// TwinCAT 3 PLC project VacuumPLC
// ProgramVersion: 3.1.4024.0
// libraries:
//   Tc2_Standard, * (Beckhoff Automation GmbH)
//   Tc2_System, * (Beckhoff Automation GmbH)
//   Tc3_Module, * (Beckhoff Automation GmbH)
// project tree:
//   DUTs/ Loader.TcDUT, Pump.TcDUT
//   GVLs/ GVL.TcGVL
//   / PlcTask.TcTTO
//   POUs/ Alarms.TcPOU, Common_Pulses.TcPOU, HMI.TcPOU, MAIN.TcPOU, Loaders.TcPOU, Pumps.TcPOU
//   POUs/Blocks and Functions/ BitCounter.TcPOU (not stored), FB_Loader.TcPOU
// real-time tasks:
//   TASK PlcTask: cycle T#10ms, priority 20, ADS port 350
// I/O:
//   DEVICE Device 2 (EtherCAT), AmsNetId 192.168.250.42.3.1
//     Term 5 (EK1200) [EK1200-5000 EtherCAT Power supply (2A E-Bus)]
//       Term 6 (EL3064) [EL3064 4Ch. Ana. Input 0-10V]
//       Term 7 (EL4002) [EL4002 2Ch. Ana. Output 0-10V, 12bit]
//       Term 8 (EL1889) [EL1889 16Ch. Dig. Input 24V, 3ms, negative]
//       Term 9 (EL2889) [EL2889 16Ch. Dig. Output 24V, 0.5A, negative]
//       Term 10 (EL6021) [EL6021 Interface (RS422/485)]
//       Term 11 (EK1122) [EK1122 2 port EtherCAT junction]
//       Term 12 (EL9011) [EL9011 End Terminal]
// variable links:
//   VacuumPLC/VacuumPLC Instance <-> Device 2 (EtherCAT)/Term 5 (EK1200)/Term 8 (EL1889)
//     PlcTask Inputs/Loaders.Loader_1.Flap_Reed <-> Channel 4/Input
//     PlcTask Inputs/Loaders.Loader_1.Level_Prox <-> Channel 3/Input
//     PlcTask Inputs/Loaders.Loader_1.Switch <-> Channel 5/Input
//     PlcTask Inputs/Pumps.Pump_1.Over_Load <-> Channel 2/Input
//     PlcTask Inputs/Pumps.Pump_1.Switch <-> Channel 1/Input
//   VacuumPLC/VacuumPLC Instance <-> Device 2 (EtherCAT)/Term 5 (EK1200)/Term 9 (EL2889)
//     PlcTask Outputs/Loaders.Loader_1.Valve <-> Channel 7/Output
//     PlcTask Outputs/Pumps.Pump_1.Join_Valve <-> Channel 6/Output
//     PlcTask Outputs/Pumps.Pump_1.Lamp <-> Channel 1/Output
//     PlcTask Outputs/Pumps.Pump_1.Line_Block <-> Channel 5/Output
//     PlcTask Outputs/Pumps.Pump_1.Motor <-> Channel 2/Output
//     PlcTask Outputs/Pumps.Pump_1.Pump_Block <-> Channel 3/Output
//     PlcTask Outputs/Pumps.Pump_1.Pump_Vent <-> Channel 4/Output

CONFIGURATION VacuumPLC
    RESOURCE PLC ON TwinCAT3
        TASK PlcTask(INTERVAL := T#10ms, PRIORITY := 20);
        PROGRAM MAIN WITH PlcTask : MAIN;
    END_RESOURCE
END_CONFIGURATION

// ---- DUTs/Loader.TcDUT
TYPE Loader :
STRUCT
	Level_Prox AT%I* : BOOL;
	Flap_Reed AT%I* : BOOL;
	Switch AT%I* : BOOL;
	PushButton AT%I* : BOOL;
	Valve AT%Q* : BOOL;
	Lamp AT%Q* : BOOL;
	Status_Word : WORD;
	HMI_Status_Word : WORD;
END_STRUCT
END_TYPE

// ---- DUTs/Pump.TcDUT
TYPE Pump :
STRUCT
	Switch AT%I* : BOOL;
	Over_Load AT%I* : BOOL;
	Lamp AT%Q* : BOOL;
	Motor AT%Q* : BOOL;
	Pump_Block AT%Q* : BOOL;
	Pump_Vent AT%Q* : BOOL;
	Line_Block AT%Q* : BOOL;
	Join_Valve AT%Q* : BOOL;
	{attribute 'OPC.UA.DA' := '1'}
	Status_Word : WORD;
	Rest_Time : CTU;
	Off_Delay : TON;
	Clean_On : CTU;
	Air_Delay : TON;
	Steady : TON;
	Conv_End : CTU;
	Max_Conv_Time : TON;
	Max_Conv_Time_ET : TIME;
	Min_Conv_Time : TON;
	Accumulated_Time : DINT;
	Efficency : INT;
	Temp_Accum_Time : INT;
	Locel_Request : BOOL;
	Global_Request : BOOL;
	Global_Grant : BOOL;
	Line_Live : BOOL;
	Locked_1 : BOOL;
	Locked_2 : BOOL;
	START_Conv : BOOL;
	LOCK_Start : BOOL;
	AUTO_Clean : BOOL;
	PumpOnDifu  : BOOL;
	Top_prox_OK : BOOL;
	Auto_Clean_Keep : SR;
	Pump_Block_Keep : SR;
	Locked_2_Keep : RS;
	Motor_Keep : RS;
	Scanner : INT;
	Pump_Requests : INT;
	Lock_Start_DIFU : R_TRIG;
	Conv_Start_DIFU : R_TRIG;
	Max_Conv_Time_PT : TIME; 
	Vac_Req_Sum : UINT;
	Vac_Req_Size : UINT := 32;
	Clean_Delay_PV : UINT := 300; //Use this VAR to be able to change when needs to initiate auto clean before shot down
	Clean_Delay_CV : INT := 300;
	Clean_Delay_Keep : SR;
	Clean_Delay_DIFU : R_TRIG;
END_STRUCT
END_TYPE

// ---- GVLs/GVL.TcGVL
//{attribute 'qualified_only'}
VAR_GLOBAL
	Always_ON : BOOL := 1;
	Vacuum_Grants : ARRAY [0..31] OF BOOL;
	Vacuum_Requests : ARRAY [0..31] OF BOOL;
	Conv_Max_Times : ARRAY [0..31] OF DWORD := [32(30000)];
	Conv_Last_Times : ARRAY [0..31] OF DWORD;
	testvar : WORD;
END_VAR

// ---- POUs/MAIN.TcPOU
PROGRAM MAIN
VAR
END_VAR

// To activate a section in the progem it has to be written in the MAIN (PRG). the sequence of the sections would determine what run first in the progrem.
Common_Pulses();
Pumps();
Loaders();
Alarms();
	GVL.testvar := Pumps.Pump_1.Status_Word;

END_PROGRAM

// ---- POUs/Common_Pulses.TcPOU
PROGRAM Common_Pulses
VAR
	Timer_0_1_s : TON;		// 0.1 seconds pulse
	Timer_1_0_s : TON;		// 1.0 seconds pulse
	Timer_1_0_m : TON;		// 1.0 minutes pulse
	Timer_10_0_m : TON;		// 10.0 minutes pulse
	Timer0_5_s_ON : TON;	// 0.5 second TON for 1 second blink like P_1_0 from CJ
	Timer0_5_s_OFF : TOF;	// 0.5 second TOF for 1 second blink like P_1_0 from CJ
	Timer_50_ms_ON : TON;	// 50 mili second TON for 0.1 second blink like P_0_1 from CJ
	Timer_50_ms_OFF : TOF;	// 50 mili second TOF for 0.1 second blink like P_0_1 from CJ
	Blink_1_s : BOOL;		// 1 second blink for lamp when ON
	Blink_0_1_s : BOOL;		// 0.1 second blink for lamp when alarm
END_VAR

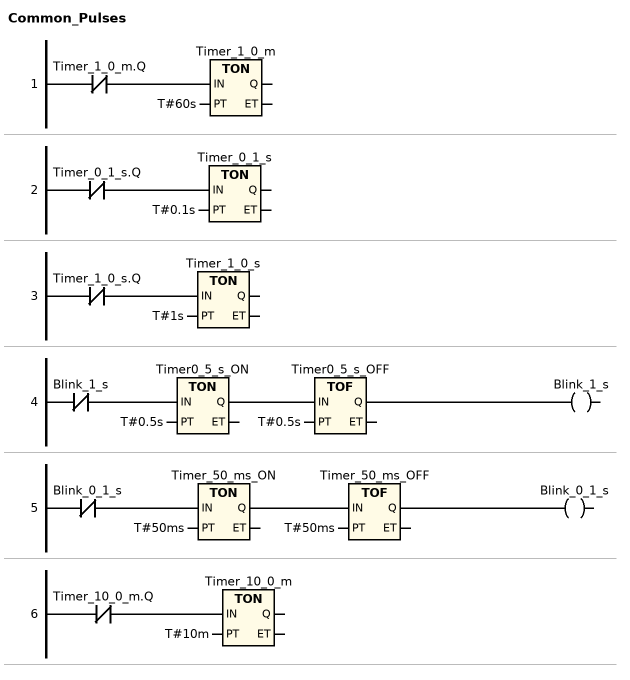
// NETWORK 1
Timer_1_0_m(IN := NOT Timer_1_0_m.Q, PT := T#60s); // TON

// NETWORK 2
Timer_0_1_s(IN := NOT Timer_0_1_s.Q, PT := T#0.1s); // TON

// NETWORK 3
Timer_1_0_s(IN := NOT Timer_1_0_s.Q, PT := T#1s); // TON

// NETWORK 4
Timer0_5_s_ON(IN := NOT Blink_1_s, PT := T#0.5s); // TON
Timer0_5_s_OFF(IN := Timer0_5_s_ON.Q, PT := T#0.5s); // TOF
Blink_1_s := Timer0_5_s_OFF.Q;

// NETWORK 5
Timer_50_ms_ON(IN := NOT Blink_0_1_s, PT := T#50ms); // TON
Timer_50_ms_OFF(IN := Timer_50_ms_ON.Q, PT := T#50ms); // TOF
Blink_0_1_s := Timer_50_ms_OFF.Q;

// NETWORK 6
Timer_10_0_m(IN := NOT Timer_10_0_m.Q, PT := T#10m); // TON

END_PROGRAM

// ---- POUs/Pumps.TcPOU
PROGRAM Pumps
VAR
	Pump_1 : Pump;
END_VAR
VAR // added by the converter: edge detectors and wires of the graphical bodies
    _w1, _w2, _w3, _w4, _w5, _w6, _w7, _w8, _w9 : BOOL;
END_VAR

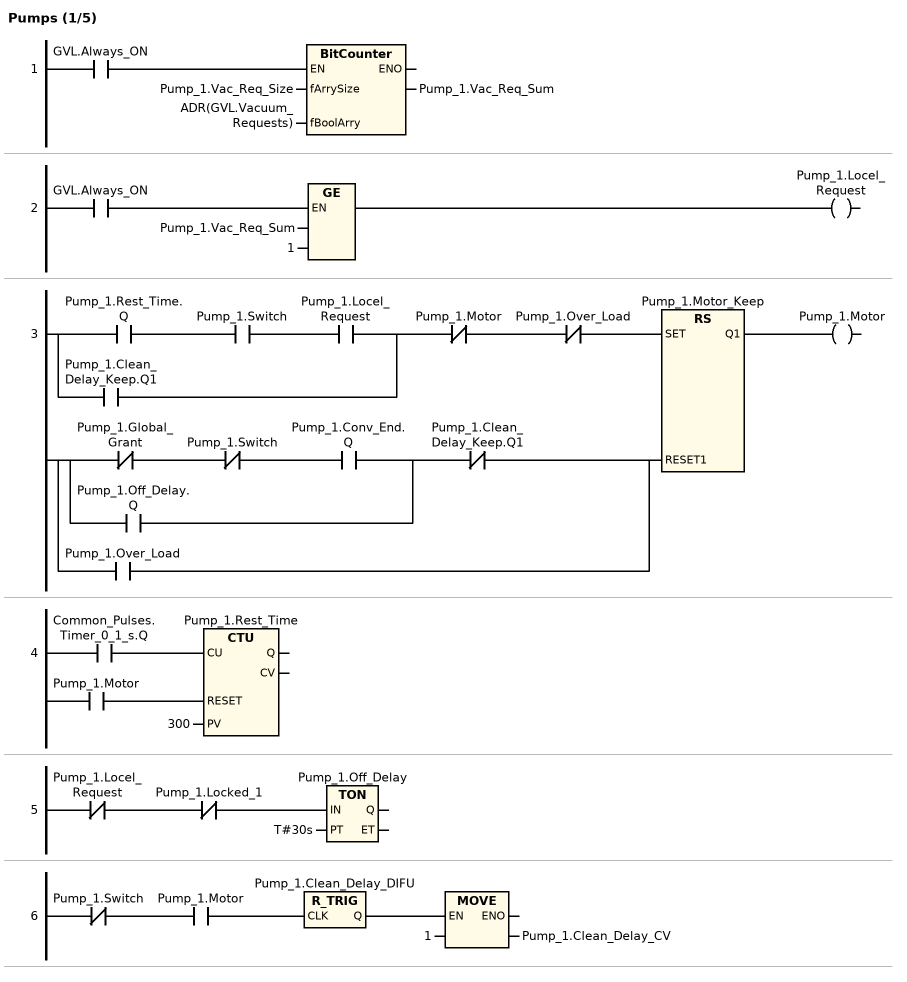
// NETWORK 1
IF GVL.Always_ON THEN
    Pump_1.Vac_Req_Sum := BitCounter(fArrySize := Pump_1.Vac_Req_Size, fBoolArry := ADR(GVL.Vacuum_Requests));
END_IF

// NETWORK 2
Pump_1.Locel_Request := GVL.Always_ON AND Pump_1.Vac_Req_Sum >= 1;

// NETWORK 3
Pump_1.Motor_Keep(SET := (Pump_1.Rest_Time.Q AND Pump_1.Switch AND Pump_1.Locel_Request OR Pump_1.Clean_Delay_Keep.Q1) AND NOT Pump_1.Motor AND NOT Pump_1.Over_Load, RESET1 := (NOT Pump_1.Global_Grant AND NOT Pump_1.Switch AND Pump_1.Conv_End.Q OR Pump_1.Off_Delay.Q) AND NOT Pump_1.Clean_Delay_Keep.Q1 OR Pump_1.Over_Load); // RS
Pump_1.Motor := Pump_1.Motor_Keep.Q1;

// NETWORK 4
Pump_1.Rest_Time(CU := Common_Pulses.Timer_0_1_s.Q, RESET := Pump_1.Motor, PV := 300); // CTU

// NETWORK 5
Pump_1.Off_Delay(IN := NOT Pump_1.Locel_Request AND NOT Pump_1.Locked_1, PT := T#30s); // TON

// NETWORK 6
Pump_1.Clean_Delay_DIFU(CLK := NOT Pump_1.Switch AND Pump_1.Motor); // R_TRIG
IF Pump_1.Clean_Delay_DIFU.Q THEN Pump_1.Clean_Delay_CV := 1; END_IF

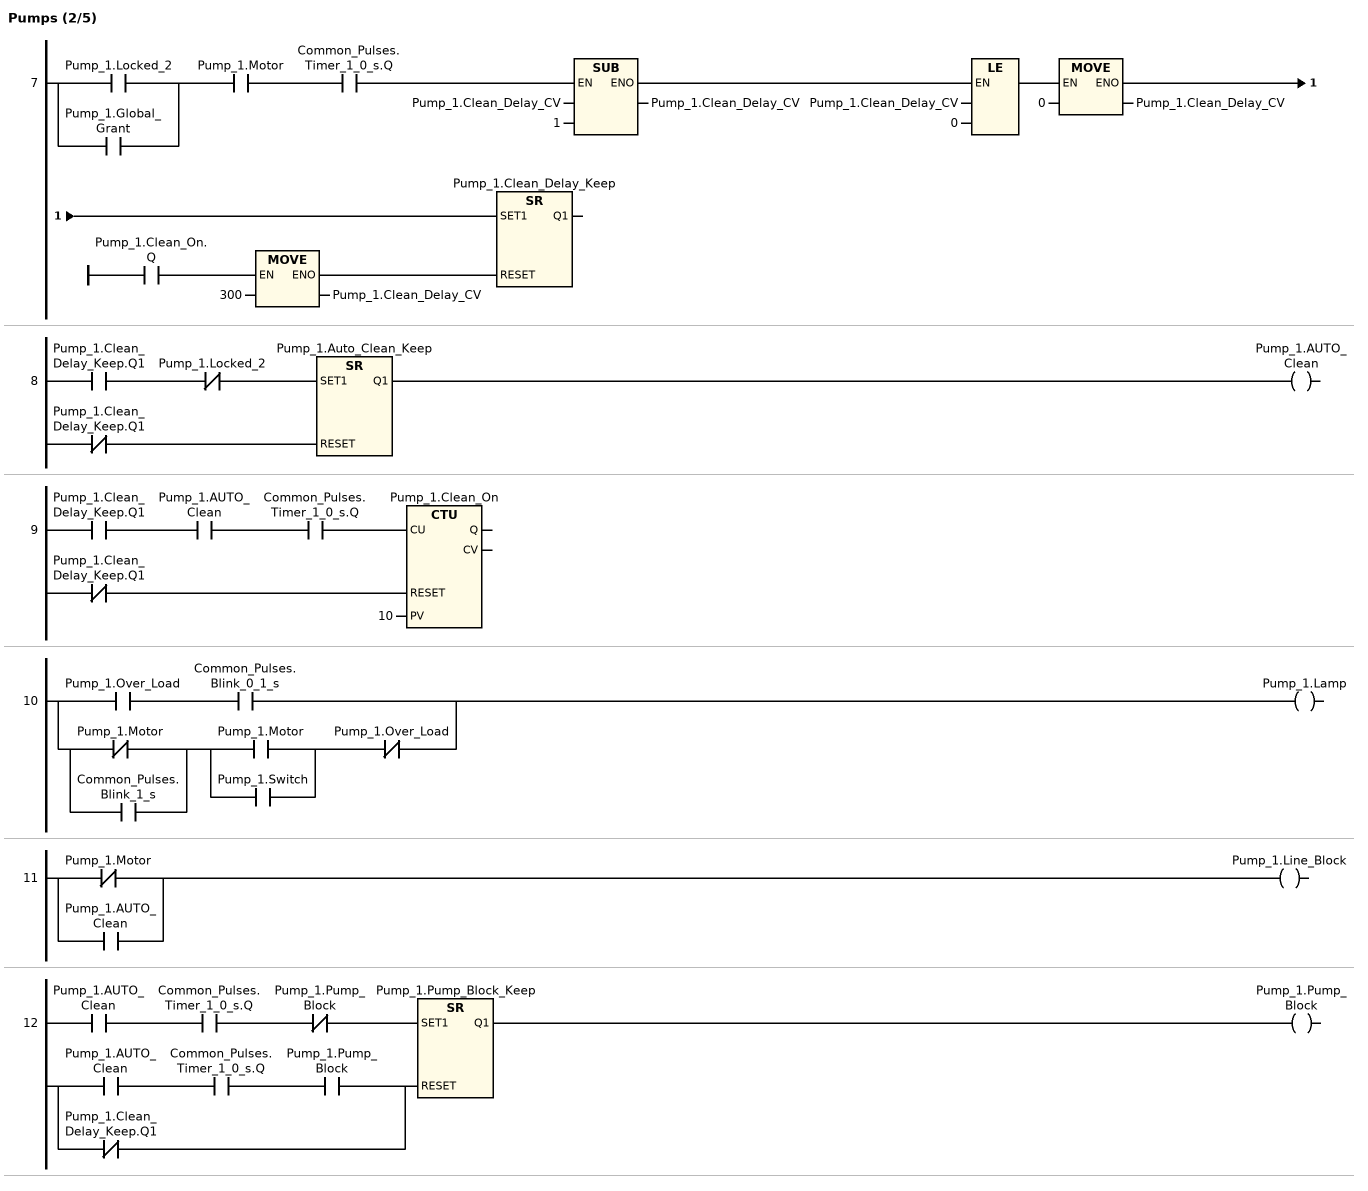
// NETWORK 7
_w1 := (Pump_1.Locked_2 OR Pump_1.Global_Grant) AND Pump_1.Motor AND Common_Pulses.Timer_1_0_s.Q;
IF _w1 THEN Pump_1.Clean_Delay_CV := Pump_1.Clean_Delay_CV - 1; END_IF
IF _w1 AND Pump_1.Clean_Delay_CV <= 0 THEN Pump_1.Clean_Delay_CV := 0; END_IF
_w3 := _w1 AND Pump_1.Clean_Delay_CV <= 0;
_w2 := Pump_1.Clean_On.Q;
IF _w2 THEN Pump_1.Clean_Delay_CV := 300; END_IF
Pump_1.Clean_Delay_Keep(SET1 := _w3, RESET := _w2); // SR

// NETWORK 8
Pump_1.Auto_Clean_Keep(SET1 := Pump_1.Clean_Delay_Keep.Q1 AND NOT Pump_1.Locked_2, RESET := NOT Pump_1.Clean_Delay_Keep.Q1); // SR
Pump_1.AUTO_Clean := Pump_1.Auto_Clean_Keep.Q1;

// NETWORK 9
Pump_1.Clean_On(
    CU := Pump_1.Clean_Delay_Keep.Q1 AND Pump_1.AUTO_Clean AND Common_Pulses.Timer_1_0_s.Q,
    RESET := NOT Pump_1.Clean_Delay_Keep.Q1,
    PV := 10); // CTU

// NETWORK 10
Pump_1.Lamp := Pump_1.Over_Load AND Common_Pulses.Blink_0_1_s OR (NOT Pump_1.Motor OR Common_Pulses.Blink_1_s) AND (Pump_1.Motor OR Pump_1.Switch) AND NOT Pump_1.Over_Load;

// NETWORK 11
Pump_1.Line_Block := NOT Pump_1.Motor OR Pump_1.AUTO_Clean;

// NETWORK 12
Pump_1.Pump_Block_Keep(SET1 := Pump_1.AUTO_Clean AND Common_Pulses.Timer_1_0_s.Q AND NOT Pump_1.Pump_Block, RESET := Pump_1.AUTO_Clean AND Common_Pulses.Timer_1_0_s.Q AND Pump_1.Pump_Block OR NOT Pump_1.Clean_Delay_Keep.Q1); // SR
Pump_1.Pump_Block := Pump_1.Pump_Block_Keep.Q1;

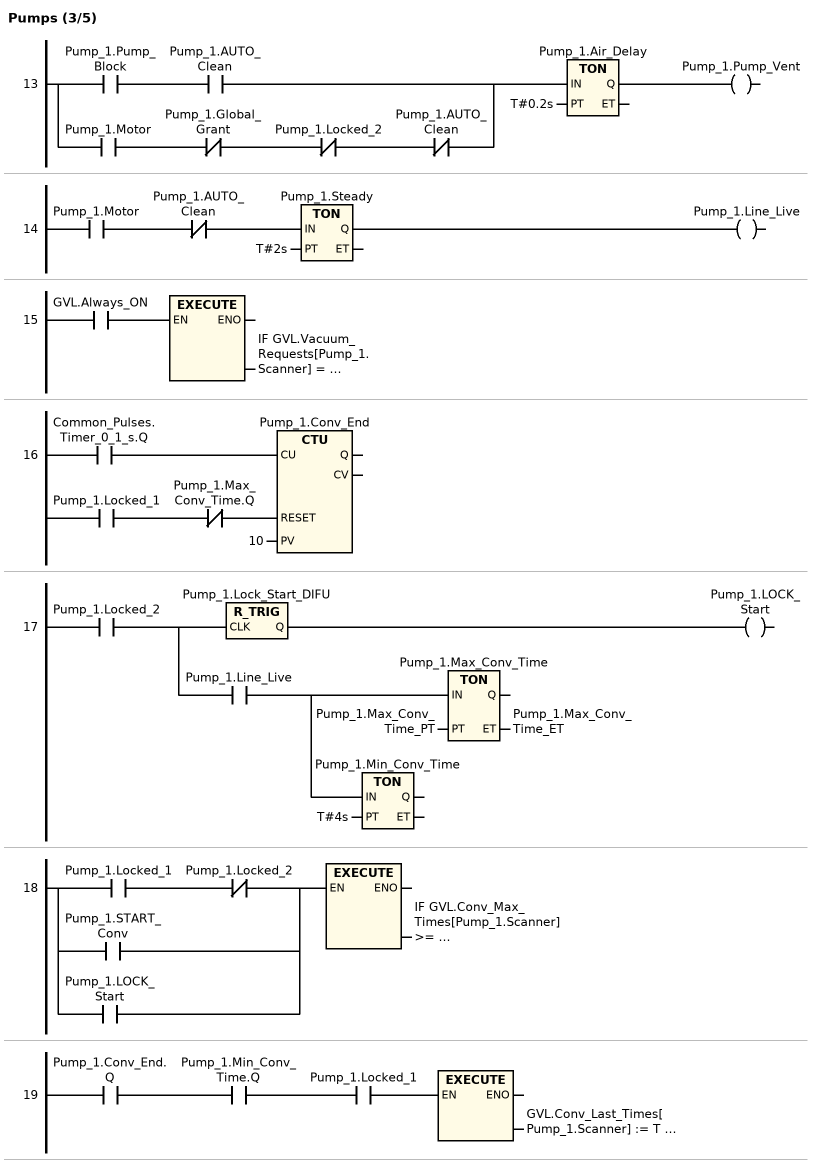
// NETWORK 13
Pump_1.Air_Delay(IN := Pump_1.Pump_Block AND Pump_1.AUTO_Clean OR Pump_1.Motor AND NOT Pump_1.Global_Grant AND NOT Pump_1.Locked_2 AND NOT Pump_1.AUTO_Clean, PT := T#0.2s); // TON
Pump_1.Pump_Vent := Pump_1.Air_Delay.Q;

// NETWORK 14
Pump_1.Steady(IN := Pump_1.Motor AND NOT Pump_1.AUTO_Clean, PT := T#2s); // TON
Pump_1.Line_Live := Pump_1.Steady.Q;

// NETWORK 15
IF GVL.Always_ON THEN
    IF GVL.Vacuum_Requests[Pump_1.Scanner] = 1 THEN 
    	Pump_1.Locked_1 := TRUE;
    	ELSE Pump_1.Locked_1 := FALSE;
    END_IF
END_IF

// NETWORK 16
Pump_1.Conv_End(
    CU := Common_Pulses.Timer_0_1_s.Q,
    RESET := Pump_1.Locked_1 AND NOT Pump_1.Max_Conv_Time.Q,
    PV := 10); // CTU

// NETWORK 17
Pump_1.Lock_Start_DIFU(CLK := Pump_1.Locked_2); // R_TRIG
Pump_1.LOCK_Start := Pump_1.Lock_Start_DIFU.Q;
_w4 := Pump_1.Locked_2 AND Pump_1.Line_Live;
Pump_1.Max_Conv_Time(IN := _w4, PT := Pump_1.Max_Conv_Time_PT, ET => Pump_1.Max_Conv_Time_ET); // TON
Pump_1.Min_Conv_Time(IN := _w4, PT := T#4s); // TON

// NETWORK 18
IF Pump_1.Locked_1 AND NOT Pump_1.Locked_2 OR Pump_1.START_Conv OR Pump_1.LOCK_Start THEN
    IF GVL.Conv_Max_Times[Pump_1.Scanner] >= 5000 THEN
    	Pump_1.Max_Conv_Time_PT := DWORD_TO_TIME(GVL.Conv_Max_Times[Pump_1.Scanner]);
    	ELSE Pump_1.Max_Conv_Time.PT := T#5S;
    END_IF
END_IF

// NETWORK 19
IF Pump_1.Conv_End.Q AND Pump_1.Min_Conv_Time.Q AND Pump_1.Locked_1 THEN
    GVL.Conv_Last_Times[Pump_1.Scanner] := TIME_TO_DWORD(Pump_1.Max_Conv_Time.ET);
    MEMSET (destAddr := ADR(GVL.Vacuum_Requests), fillByte := 0, n := SIZEOF(GVL.Vacuum_Requests));
END_IF

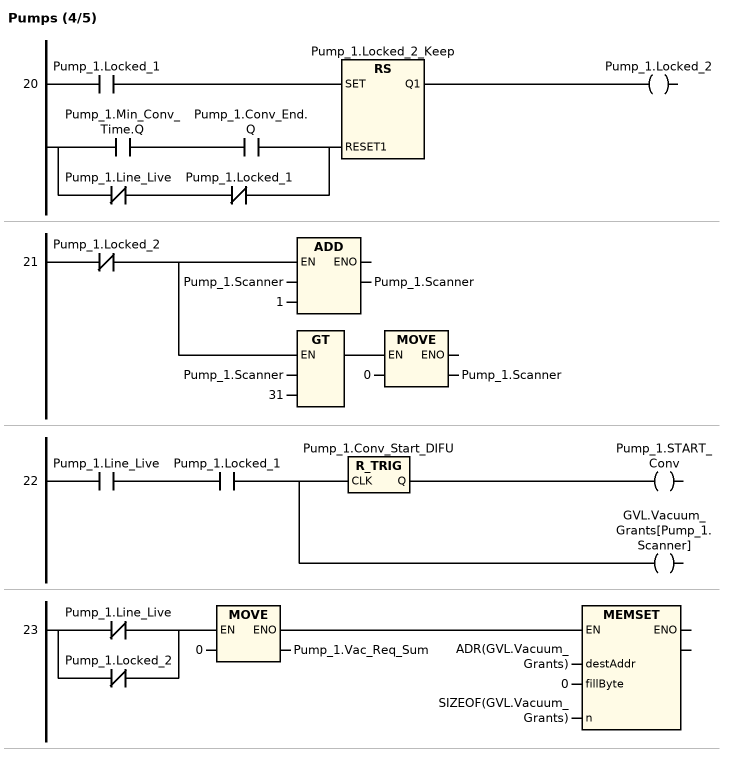
// NETWORK 20
Pump_1.Locked_2_Keep(SET := Pump_1.Locked_1, RESET1 := Pump_1.Min_Conv_Time.Q AND Pump_1.Conv_End.Q OR NOT Pump_1.Line_Live AND NOT Pump_1.Locked_1); // RS
Pump_1.Locked_2 := Pump_1.Locked_2_Keep.Q1;

// NETWORK 21
_w5 := NOT Pump_1.Locked_2;
IF _w5 THEN Pump_1.Scanner := Pump_1.Scanner + 1; END_IF
IF _w5 AND Pump_1.Scanner > 31 THEN Pump_1.Scanner := 0; END_IF

// NETWORK 22
_w6 := Pump_1.Line_Live AND Pump_1.Locked_1;
Pump_1.Conv_Start_DIFU(CLK := _w6); // R_TRIG
Pump_1.START_Conv := Pump_1.Conv_Start_DIFU.Q;
GVL.Vacuum_Grants[Pump_1.Scanner] := _w6;

// NETWORK 23
_w7 := NOT Pump_1.Line_Live OR NOT Pump_1.Locked_2;
IF _w7 THEN Pump_1.Vac_Req_Sum := 0; END_IF
IF _w7 THEN MEMSET(destAddr := ADR(GVL.Vacuum_Grants), fillByte := 0, n := SIZEOF(GVL.Vacuum_Grants)); END_IF

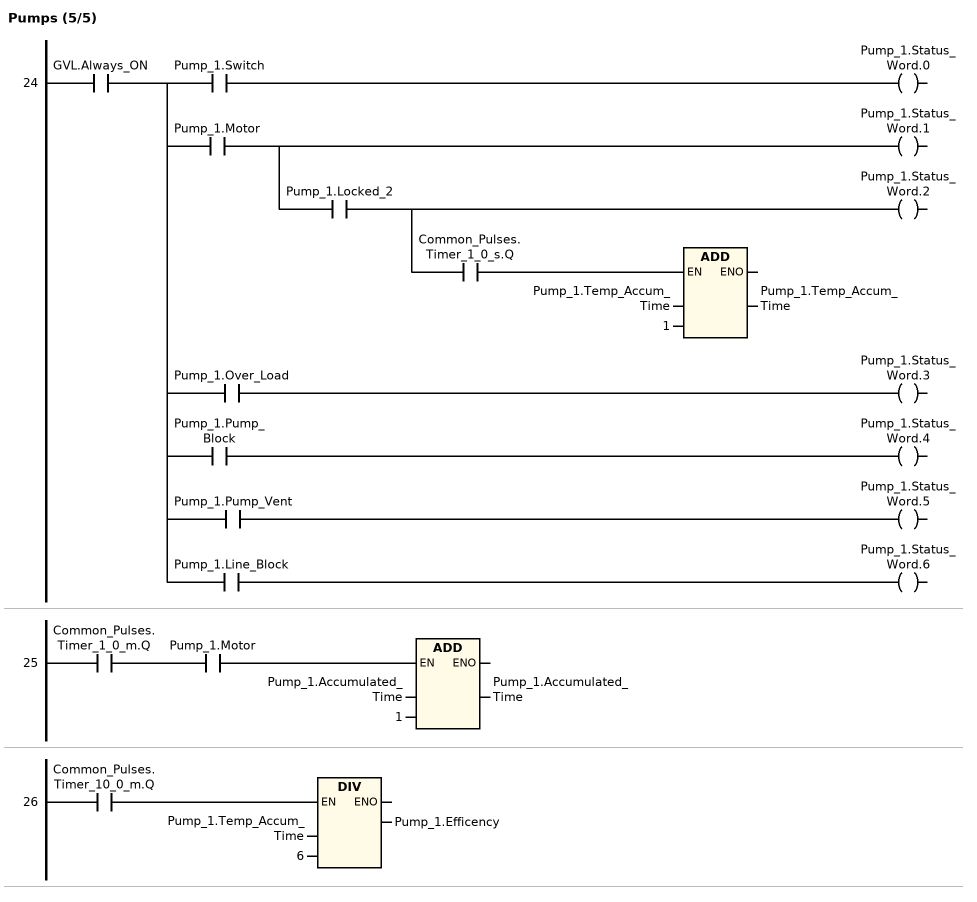
// NETWORK 24
Pump_1.Status_Word.0 := GVL.Always_ON AND Pump_1.Switch;
_w8 := GVL.Always_ON AND Pump_1.Motor;
Pump_1.Status_Word.1 := _w8;
_w9 := _w8 AND Pump_1.Locked_2;
Pump_1.Status_Word.2 := _w9;
IF _w9 AND Common_Pulses.Timer_1_0_s.Q THEN Pump_1.Temp_Accum_Time := Pump_1.Temp_Accum_Time + 1; END_IF
Pump_1.Status_Word.3 := GVL.Always_ON AND Pump_1.Over_Load;
Pump_1.Status_Word.4 := GVL.Always_ON AND Pump_1.Pump_Block;
Pump_1.Status_Word.5 := GVL.Always_ON AND Pump_1.Pump_Vent;
Pump_1.Status_Word.6 := GVL.Always_ON AND Pump_1.Line_Block;

// NETWORK 25
IF Common_Pulses.Timer_1_0_m.Q AND Pump_1.Motor THEN Pump_1.Accumulated_Time := Pump_1.Accumulated_Time + 1; END_IF

// NETWORK 26
IF Common_Pulses.Timer_10_0_m.Q THEN Pump_1.Efficency := Pump_1.Temp_Accum_Time / 6; END_IF

END_PROGRAM

// ---- POUs/Loaders.TcPOU
PROGRAM Loaders
VAR
	Loader_1: Loader;
	Loader_2: Loader;
	Loader_3: Loader;
	FB_Loader_1: FB_Loader;
	FB_Loader_2: FB_Loader;
	FB_Loader_3: FB_Loader;
END_VAR

// note: this text did not pass the execution check against the stored diagram
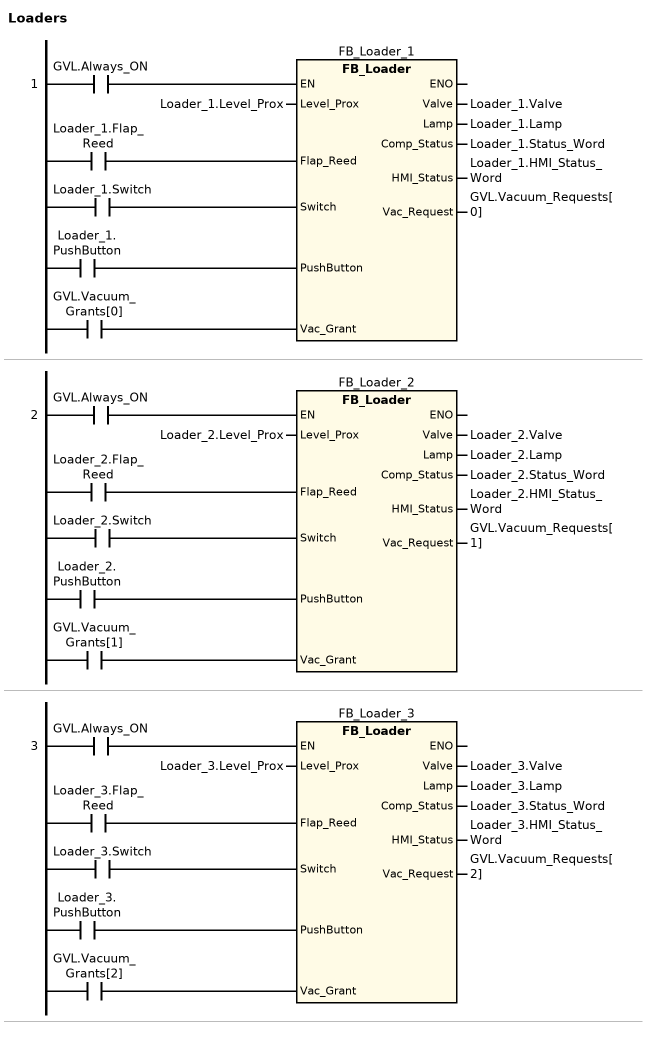
// NETWORK 1
FB_Loader_1(
    EN := GVL.Always_ON,
    Level_Prox := Loader_1.Level_Prox,
    Flap_Reed := Loader_1.Flap_Reed,
    Switch := Loader_1.Switch,
    PushButton := Loader_1.PushButton,
    Vac_Grant := GVL.Vacuum_Grants[0],
    Valve => Loader_1.Valve,
    Lamp => Loader_1.Lamp,
    Comp_Status => Loader_1.Status_Word,
    HMI_Status => Loader_1.HMI_Status_Word,
    Vac_Request => GVL.Vacuum_Requests[0]); // FB_Loader

// NETWORK 2
FB_Loader_2(
    EN := GVL.Always_ON,
    Level_Prox := Loader_2.Level_Prox,
    Flap_Reed := Loader_2.Flap_Reed,
    Switch := Loader_2.Switch,
    PushButton := Loader_2.PushButton,
    Vac_Grant := GVL.Vacuum_Grants[1],
    Valve => Loader_2.Valve,
    Lamp => Loader_2.Lamp,
    Comp_Status => Loader_2.Status_Word,
    HMI_Status => Loader_2.HMI_Status_Word,
    Vac_Request => GVL.Vacuum_Requests[1]); // FB_Loader

// NETWORK 3
FB_Loader_3(
    EN := GVL.Always_ON,
    Level_Prox := Loader_3.Level_Prox,
    Flap_Reed := Loader_3.Flap_Reed,
    Switch := Loader_3.Switch,
    PushButton := Loader_3.PushButton,
    Vac_Grant := GVL.Vacuum_Grants[2],
    Valve => Loader_3.Valve,
    Lamp => Loader_3.Lamp,
    Comp_Status => Loader_3.Status_Word,
    HMI_Status => Loader_3.HMI_Status_Word,
    Vac_Request => GVL.Vacuum_Requests[2]); // FB_Loader

END_PROGRAM

// ---- POUs/Blocks and Functions/FB_Loader.TcPOU
FUNCTION_BLOCK FB_Loader
VAR_INPUT
	EN : BOOL;
	Level_Prox : BOOL; // Loader Proximity Switch
	Flap_Reed : BOOL; // Loader Flap Reed Switch
	Switch : BOOL; // Loader switch
	PushButton : BOOL; // Loader Push Button
	Vac_Grant : BOOL; // Vacuum Grant to the Loader
	Switch_Bit : BOOL; // Loader internal Switch Bit - Push Button or Switch
END_VAR
VAR_OUTPUT
	ENO : BOOL;
	Valve : BOOL; // Loader Vacuum Valve
	Lamp : BOOL; // Loader status lamp
	Comp_Status : WORD; // Loader status word for Sysmetric Vision
	HMI_Status : WORD; // Loader status word for HMI
	Vac_Request : BOOL; // Vacuum Request from the loader
END_VAR
VAR
	Timer_0_1 : TON;		// 0.1 seconds timer for counters
	Timer0_5_s_ON : TON;	// 0.5 second TON for 1 second blink like P_1_0 from CJ
	Timer0_5_s_OFF : TOF;	// 0.5 second TOF for 1 second blink like P_1_0 from CJ
	Timer_50_ms_ON : TON;	// 50 mili second TON for 0.1 second blink like P_0_1 from CJ
	Timer_50_ms_OFF : TOF;	// 50 mili second TOF for 0.1 second blink like P_0_1 from CJ
	MATfallTIME : CTU;		// Material fall time after conveying usually 8 seconds
	Flap_Open_time : CTU;	// check if Flap is open for more than 1.5 second, if true cancel conveying alarm
	CONValarm : CTU;		// conveying alarm turn on after usually 4 bad conveyings
	One_Time : BOOL;		// allow a loader on dosing system to request conveying only one per vacuum grant from main PLC
	Switch_Keep : SR;		// Conveying Push botton switch
	Blink_1_0_s: BOOL;		// 1 second blink for loaders lamp when ON
	Blink_0_1_s: BOOL;		// 0.1 second blink for loaders lamp when alarm
END_VAR
VAR // added by the converter: edge detectors and wires of the graphical bodies
    _rt1, _rt2 : R_TRIG;
    _ft1 : F_TRIG;
    _w1, _w2, _w3 : BOOL;
END_VAR

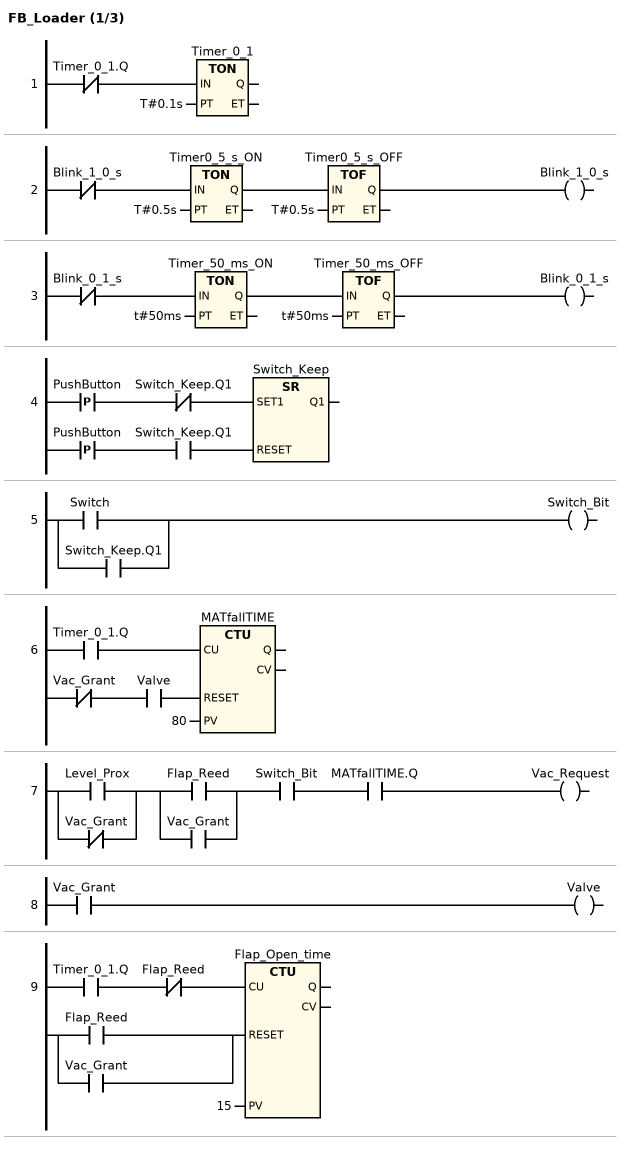
// NETWORK 1
Timer_0_1(IN := NOT Timer_0_1.Q, PT := T#0.1s); // TON

// NETWORK 2
Timer0_5_s_ON(IN := NOT Blink_1_0_s, PT := T#0.5s); // TON
Timer0_5_s_OFF(IN := Timer0_5_s_ON.Q, PT := T#0.5s); // TOF
Blink_1_0_s := Timer0_5_s_OFF.Q;

// NETWORK 3
Timer_50_ms_ON(IN := NOT Blink_0_1_s, PT := t#50ms); // TON
Timer_50_ms_OFF(IN := Timer_50_ms_ON.Q, PT := t#50ms); // TOF
Blink_0_1_s := Timer_50_ms_OFF.Q;

// NETWORK 4
_rt1(CLK := PushButton);
_rt2(CLK := PushButton);
Switch_Keep(SET1 := _rt1.Q AND NOT Switch_Keep.Q1, RESET := _rt2.Q AND Switch_Keep.Q1); // SR

// NETWORK 5
Switch_Bit := Switch OR Switch_Keep.Q1;

// NETWORK 6
MATfallTIME(CU := Timer_0_1.Q, RESET := NOT Vac_Grant AND Valve, PV := 80); // CTU

// NETWORK 7
Vac_Request := (Level_Prox OR NOT Vac_Grant) AND (Flap_Reed OR Vac_Grant) AND Switch_Bit AND MATfallTIME.Q;

// NETWORK 8
Valve := Vac_Grant;

// NETWORK 9
Flap_Open_time(CU := Timer_0_1.Q AND NOT Flap_Reed, RESET := Flap_Reed OR Vac_Grant, PV := 15); // CTU

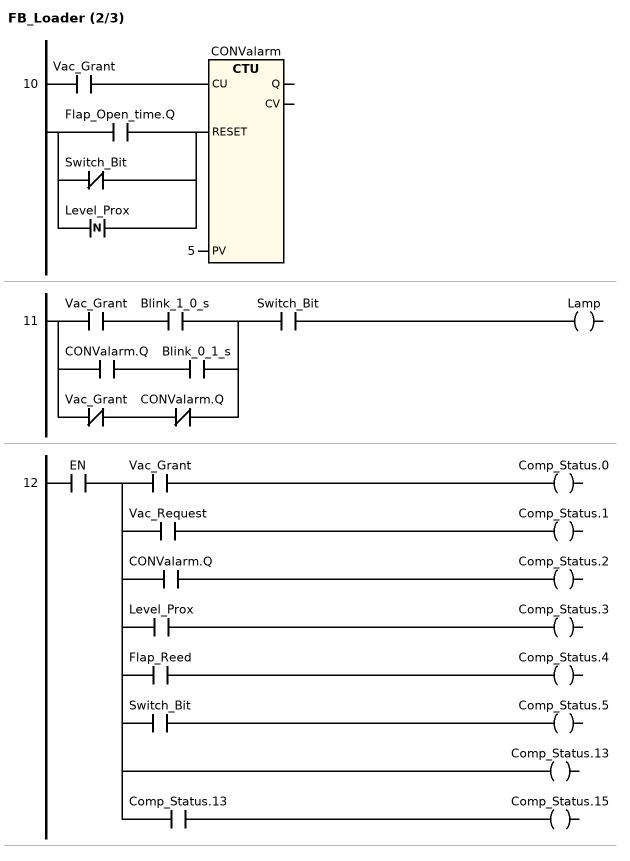
// NETWORK 10
_ft1(CLK := Level_Prox);
CONValarm(CU := Vac_Grant, RESET := Flap_Open_time.Q OR NOT Switch_Bit OR _ft1.Q, PV := 5); // CTU

// NETWORK 11
Lamp := (Vac_Grant AND Blink_1_0_s OR CONValarm.Q AND Blink_0_1_s OR NOT Vac_Grant AND NOT CONValarm.Q) AND Switch_Bit;

// NETWORK 12
Comp_Status.0 := EN AND Vac_Grant;
Comp_Status.1 := EN AND Vac_Request;
Comp_Status.2 := EN AND CONValarm.Q;
Comp_Status.3 := EN AND Level_Prox;
Comp_Status.4 := EN AND Flap_Reed;
Comp_Status.5 := EN AND Switch_Bit;
Comp_Status.13 := EN;
Comp_Status.15 := EN AND Comp_Status.13;

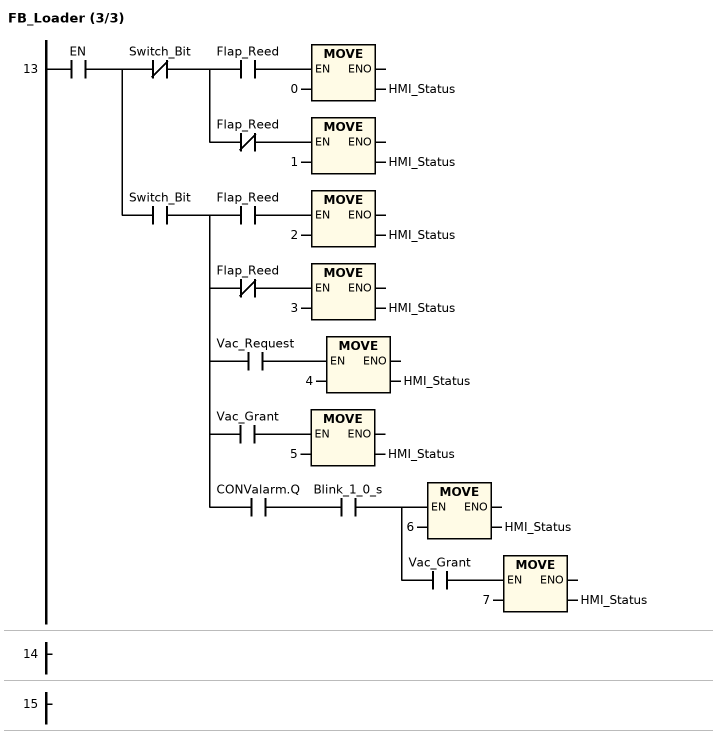
// NETWORK 13
_w1 := EN AND NOT Switch_Bit;
IF _w1 AND Flap_Reed THEN HMI_Status := 0; END_IF
IF _w1 AND NOT Flap_Reed THEN HMI_Status := 1; END_IF
_w2 := EN AND Switch_Bit;
IF _w2 AND Flap_Reed THEN HMI_Status := 2; END_IF
IF _w2 AND NOT Flap_Reed THEN HMI_Status := 3; END_IF
IF _w2 AND Vac_Request THEN HMI_Status := 4; END_IF
IF _w2 AND Vac_Grant THEN HMI_Status := 5; END_IF
_w3 := _w2 AND CONValarm.Q AND Blink_1_0_s;
IF _w3 THEN HMI_Status := 6; END_IF
IF _w3 AND Vac_Grant THEN HMI_Status := 7; END_IF

// NETWORK 14

// NETWORK 15

END_FUNCTION_BLOCK

// ---- POUs/Alarms.TcPOU
PROGRAM Alarms
VAR
	Alarms_Array : ARRAY [0..255] OF BOOL; 	//this is the alarms array for all the alarms of a given system. if a larger arry in needed eiter use to Bit Counter functions or change FOR loop in Bit Counter to much bigger array.
	Temp_AlarmCnt : UINT;					// Temp Alarm counter for active alarms check.
	AlarmCnt : UINT; 						//number of active alarms
	AlarmExist : BOOL; 						//ON as long as there is an active alarm
	Alarm_SR : SR; 							//SR replace KEEP in Omron progrem for Alarm Relay
	Alarm_Relay AT%Q* : BOOL; 				//Alarm Relay R10
	Cancel_Alarm_PB AT%I* : BOOL;			//Alarm Push Botton
END_VAR
VAR // added by the converter: edge detectors and wires of the graphical bodies
    _w1, _w2, _w3 : BOOL;
END_VAR

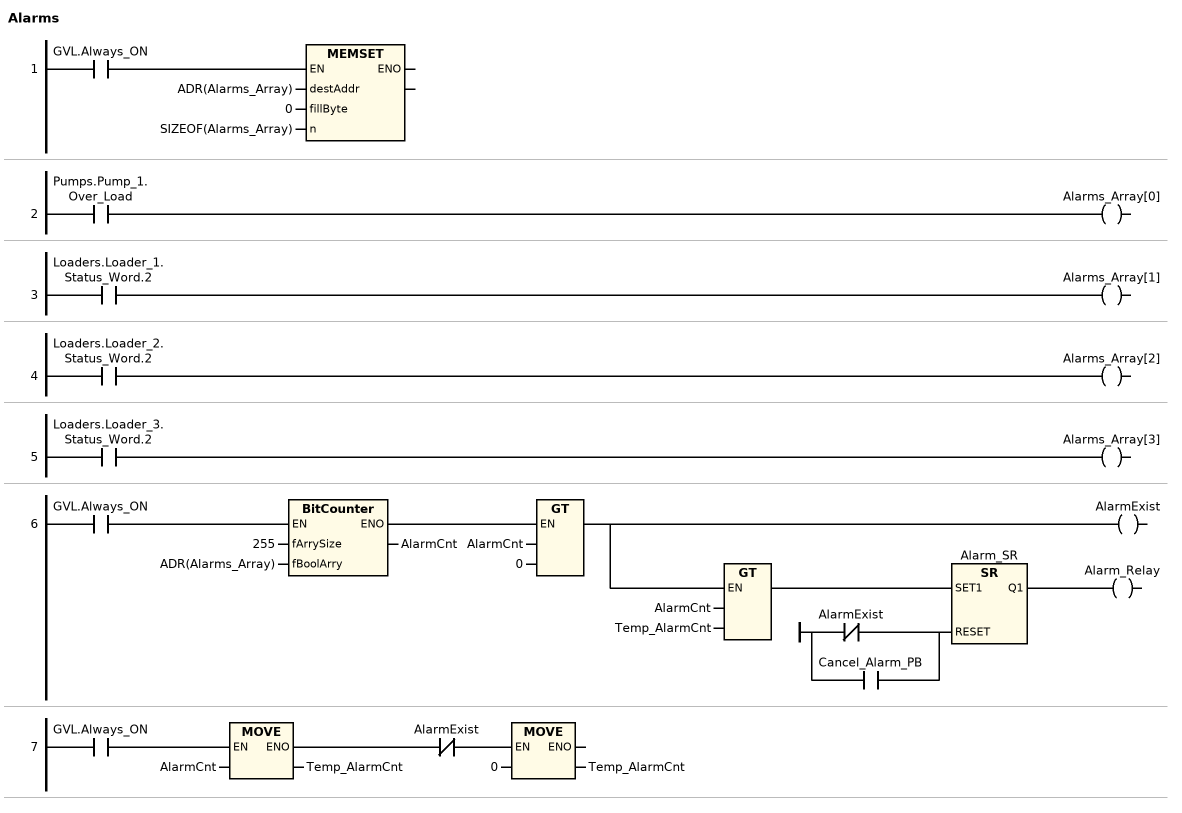
// NETWORK 1
IF GVL.Always_ON THEN MEMSET(destAddr := ADR(Alarms_Array), fillByte := 0, n := SIZEOF(Alarms_Array)); END_IF

// NETWORK 2
Alarms_Array[0] := Pumps.Pump_1.Over_Load;

// NETWORK 3
Alarms_Array[1] := Loaders.Loader_1.Status_Word.2;

// NETWORK 4
Alarms_Array[2] := Loaders.Loader_2.Status_Word.2;

// NETWORK 5
Alarms_Array[3] := Loaders.Loader_3.Status_Word.2;

// NETWORK 6
_w1 := GVL.Always_ON;
IF _w1 THEN AlarmCnt := BitCounter(fArrySize := 255, fBoolArry := ADR(Alarms_Array)); END_IF
_w2 := _w1 AND AlarmCnt > 0;
AlarmExist := _w2;
Alarm_SR(SET1 := _w2 AND AlarmCnt > Temp_AlarmCnt, RESET := NOT AlarmExist OR Cancel_Alarm_PB); // SR
Alarm_Relay := Alarm_SR.Q1;

// NETWORK 7
_w3 := GVL.Always_ON;
IF _w3 THEN Temp_AlarmCnt := AlarmCnt; END_IF
IF _w3 AND NOT AlarmExist THEN Temp_AlarmCnt := 0; END_IF

END_PROGRAM

// ---- POUs/HMI.TcPOU
PROGRAM HMI
VAR
	Loader_Name				: ARRAY [1..100] OF STRING;
	Loader_Number			: ARRAY [1..100] OF WORD;
	Loader_Status			: ARRAY [1..100] OF WORD;
	Loader_HMI_Status		: ARRAY [1..100] OF WORD;
	Loader_Last_Time		: ARRAY [1..100] OF WORD;
	Loader_Prop				: ARRAY [1..100] OF WORD;
END_VAR

// NETWORK 1

END_PROGRAM
